PROGRAM MAIN
VAR
    someInt1 : INT := 20;
	someInt2 : INT := 10;
	result : INT;
	
	bigNum : INT;
	smallNum : INT;
	
	isCaluculated : BOOL := FALSE;
	isCompared : BOOL := FALSE;
	isIncreased : BOOL := FALSE;
	
	//timers
	//set timer for 3s
	fbTon : TON := (PT:=T#3S);
	trigger : BOOL := TRUE;
	isTimerDone : BOOL := FALSE;
END_VAR

IF NOT isCaluculated THEN
	result := sum(num1 := someInt1, num2 := someInt2);
	isCaluculated := TRUE;
END_IF

IF NOT isCompared THEN
	complicatedFunc(num1:=someInt1, num2:=someInt2, biggerNum=>bigNum, smallerNum=>smallNum);
	isCompared := TRUE;	
END_IF

IF NOT isIncreased THEN
	funcWithReferences(someInt1);
	isIncreased := TRUE;	
END_IF

//timers
//start timer when trigger is true
fbTon(IN:=trigger);
isTimerDone := fbTon.Q;

END_PROGRAM

(* stored: Version 1.1.0.1, ProductVersion 3.1.4024.11
   POU MAIN: Id {3a6d0614-4b7c-4594-991a-52d589f5f757}, SpecialFunc None *)
